FUNCTION_BLOCK FB_Dog EXTENDS FB_Animal
VAR_INPUT
END_VAR
VAR_OUTPUT
END_VAR
VAR
END_VAR

METHOD M_Bark
VAR_INPUT
END_VAR
THIS^.sOutput := 'Dog barks';
END_METHOD

METHOD M_Eat
// Overrides FB_Animal's eat() — exactly like @Override in Java
THIS^.sOutput := 'Dog eats dog food';
END_METHOD

END_FUNCTION_BLOCK

(* stored: Version 1.1.0.1, ProductVersion 3.1.4024.16
   POU FB_Dog: Id {f9097222-8289-4bef-9e78-6409fca2889d}, SpecialFunc None
   Method M_Bark: Id {4e64948e-6881-450f-94f6-f2eae696d46f}
   Method M_Eat: Id {25a8afe3-5874-406b-b599-d82cd313fd78} *)
